// TIA Portal V16 export
// export: Created 2021-03-04T22:04:04.3689655Z, ExportSetting WithDefaults, DisplayName Totally Integrated Automation Portal, DisplayVersion V16, DisplayName TIA Portal Version Control Interface, DisplayVersion V16, DisplayName TIA Portal Openness, DisplayVersion V16, DisplayName SINAMICS Startdrive Advanced, DisplayVersion V16, DisplayName SINAMICS Startdrive G130, G150, S120, S150, SINAMICS MV, S210, DisplayVersion V16, DisplayName SINAMICS Startdrive G110M, G120, G120C, G120D, G120P, DisplayVersion V16, DisplayName STEP 7 Professional, DisplayVersion V16, DisplayName STEP 7 Safety, DisplayVersion V16, DisplayName WinCC Professional, DisplayVersion V16
VAR_GLOBAL   // PLC tag table "Library Constants"
END_VAR
VAR_GLOBAL CONSTANT   // user constants
   eSTATE_MANUAL : Int := 2;   // State Machine enumeration
   ePBLT_FLASHING_ENABLED : Int := 4;   // HMI PB LT enumeration
   eSTATE_RETRACTING : Int := 5;   // State Machine enumeration
   "IoScaling.S7Analog.Ni100.rScaledMax" : Real := 250.0;
   "IoScaling.S7Analog.Ni100.Climate.rScaledMax" : Real := 250.0;
   eSTEP_StoppingStart : Int := 4000;   // State Machine enumeration
   eSTEP_VerifyCenterComplete : Int := 7999;   // State Machine enumeration
   "IoScaling.S7Analog.150Ohms.rScaledMax" : Real := 150.0;
   "IoScaling.S7Analog.Default.bSwapBytes" : Bool := false;
   eANALOG_INPUTHIGHHIGH : Int := 102;
   eMOTION_DISABLED : Int := 4;   // Status Enumeration - Motion
   "IoScaling.S7Analog.Pt100.iRawMax" : Int := 8500;
   eSTEP_RetractingComplete : Int := 5999;   // State Machine enumeration
   eMODE_MANUAL : Int := 2;   // Mode enumeration
   eANALOG_INPUTINVALID : Int := 101;
   ePBLT_HIDDEN : Int := -1;   // HMI PB LT enumeration
   eVALVE_HOMEON : Int := 6;
   "IoScaling.S7Analog.Pt100.Climate.rScaledMin" : Real := -120.0;
   eHOME_ABS_RET_ABS : Int := 7;   // See MC_Home help for details
   eMOTION_ERROR : Int := 0;   // Status Enumeration - Motion
   ePB_MAINTAINED : Int := 1;   // HMI PB Type enumeration
   LKINCTRL_LENGTH_OF_PATHDATA_NAME : Int := 10;
   LKINCTRL_NO_OF_PATHDATA_ELEMENTS : Int := 15;
   "IoScaling.S7Analog.Pt100.Climate.iRawMax" : Int := 13000;
   eVALVE_ERROR : Int := 2;
   "IoScaling.S7Analog.Types.Pt100.Climate" : Int := 3;
   eMODE_INDEPENDENT : Int := 10;   // Mode
   "IoScaling.S7Analog.600Ohms.rScaledMax" : Real := 600.0;
   eMOTION_RUNNING : Int := 2;   // Status Enumeration - Motion
   "IoScaling.S7Analog.Ni100.Climate.rScaledMin" : Real := -60.0;
   eMOTION_STOPPED : Int := 1;   // Status Enumeration - Motion
   eMOTION_MAINTENANCE : Int := 3;   // Status Enumeration - Motion
   "IoScaling.S7Analog.Ni100.rScaledMin" : Real := -60.0;
   eSTATE_STOPPING : Int := 4;   // State Machine enumeration
   "IoScaling.S7Analog.Pt100.Climate.rScaledMax" : Real := 130.0;
   "IoScaling.S7Analog.Pt100.rScaledMax" : Real := 850.0;
   "IoScaling.S7Analog.Types.Ni100.Climate" : Int := 5;
   ePB_UNLATCH : Int := 3;   // HMI PB Type enumeration
   "IoScaling.S7Analog.Ni100.Climate.iRawMax" : Int := 25000;
   eSTEP_BladeChangeStart : Int := 6000;   // State Machine enumeration
   "IoScaling.S7Analog.300Ohms.rScaledMin" : Real := 0.0;
   "IoScaling.S7Analog.Types.Pt100" : Int := 2;
   LKINCTRL_PI : LReal := 3.1415926535897932846264;
   eVALVE_WORKPOSITION : Int := 3;
   eCAM_SYNCDIRECTION_SHORTESTWAY : Int := 3;   // See MC_CamIn help for details
   "IoScaling.S7Analog.Types.+-V/mA" : Int := 1;
   ePBLT_FLASHING_DISABLED : Int := 5;   // HMI PB LT enumeration
   "IoScaling.S7Analog.150Ohms.rScaledMin" : Real := 0.0;
   eHOME_ACCEPT_CURRENT : Int := 11;   // Used when the configured and current encoders don't match
   LKINCTRL_NO_OF_START_EXECUTE_CMDS : Int := 5;
   ePBLT_TRANSITIONING : Int := 2;   // HMI PB LT enumeration
   SM_ACTIVE_DYNAMICS : Int := 0;
   eVALVE_WORKON : Int := 5;
   "IoScaling.S7Analog.+-V/mA.iRawMax" : Int := 27648;
   eSTATE_INITIALIZATION : Int := 1;   // State Machine enumeration
   LKINCTRL_NO_OF_PATHDATA_PREBUFFER_ELEMENTS : Int := 5;
   eHOME_ABS_RET_OFFSET : Int := 6;   // See MC_Home help for details
   eSTEP_BladeChangeComplete : Int := 6999;   // State Machine enumeration
   eSTEP_RunningComplete : Int := 3999;   // State Machine enumeration
   eANALOG_READY : Int := 100;
   ePBLT_ENABLED : Int := 1;   // HMI PB LT enumeration
   "IoScaling.S7Analog.Pt100.Climate.iRawMin" : Int := -12000;
   eSTATE_RUNNING : Int := 3;   // State Machine enumeration
   LKINCTRL_NO_OF_LAST_FLAG : Int := 15;
   "IoScaling.S7Analog.Ni100.iRawMax" : Int := 2500;
   "IoScaling.S7Analog.Types.Default" : Int := 0;
   eHOME_ACCEPT_CONFIG : Int := 12;   // Used when the configured and current encoders don't match
   eSTEP_RunningStart : Int := 3000;   // State Machine enumeration
   "IoScaling.S7Analog.Default.iRawMin" : Int := 0;
   ePBLT_ACTIVE : Int := 3;   // HMI PB LT enumeration
   "IoScaling.S7Analog.Types.Ni100" : Int := 4;
   eMODE_AUTO : Int := 1;   // Mode enumeration
   "IoScaling.S7Analog.Default.iRawMax" : Int := 27648;
   ePBLT_DISABLED : Int := 0;   // HMI PB LT enumeration
   LKINCTRL_NO_OF_SEQ_EXECUTE_CMDS : Int := 5;
   eSTEP_StoppingComplete : Int := 4999;   // State Machine enumeration
   "IoScaling.S7Analog.Ni100.Climate.iRawMin" : Int := -6000;
   "IoScaling.S7Analog.Pt100.iRawMin" : Int := -2000;
   ePB_LATCH : Int := 2;   // HMI PB Type enumeration
   eVALVE_ESTOP : Int := 1;
   eSTEP_RetractingStart : Int := 5000;   // State Machine enumeration
   "IoScaling.S7Analog.300Ohms.rScaledMax" : Real := 300.0;
   eANALOG_INPUTLOW : Int := 105;
   "IoScaling.S7Analog.Pt100.rScaledMin" : Real := -200.0;
   eSTATE_BLADECHANGE : Int := 6;   // State Machine enumeration
   "IoScaling.S7Analog.600Ohms.rScaledMin" : Real := 0.0;
   eSTATE_VERIFYCENTER : Int := 7;   // State Machine enumeration
   eVALVE_STOPPED : Int := 0;
   eCAM_SYNCPROFILEREFERENCE_LEADINGVALUEDISTANCE : Int := 1;   // See MC_CamIn help for details
   "IoScaling.S7Analog.Ni100.iRawMin" : Int := -600;
   ePB_HELD : Int := 4;   // HMI PB Type enumeration
   LKINCTRL_NO_OF_CMD_SETFLAGS : Int := 8;
   eSTEP_VerifyCenterStart : Int := 7000;   // State Machine enumeration
   eVALVE_HOMEPOSITION : Int := 4;
   eANALOG_INPUTHIGH : Int := 104;
   eANALOG_INPUTLOWLOW : Int := 103;
   "IoScaling.S7Analog.+-V/mA.iRawMin" : Int := -27648;
   ePB_MOMENTARY : Int := 0;   // HMI PB Type enumeration
   "Modes.PID.Pretuning" : Int := 1;
   "TotalizerTimeUnits.DAYS" : Int := 4;
   "HMI.Status.ForwardWork" : Int := 3;
   "FIFO.iQueueDisabled" : Int := -1;
   "Handshakes.iSize" : Int := 5;
   "Modes.Auto" : Int := 1;
   "HMI.Status.Generic1" : Int := 101;
   "Simocode.Types.DirectStarter" : Int := 1;
   "Estop.MinSetPoint" : Int := 0;
   "Simocode.Types.OverloadRelay" : Int := 0;
   "HMI.Status.SimulatedReverseHome" : Int := 8;
   "TotalizerTimeUnits.MILLISECONDS" : Int := 0;
   "HMI.Status.Generic4" : Int := 104;
   "SoftStarter.HMI.Status.EStop" : Int := 1;
   "HMI.Status.OnForwardWork" : Int := 5;
   "DataTypes.iMaxInt" : Int := 32767;
   "FIFO.iQueueSize" : Int := 5;
   "Modes.PID.ManualMode" : Int := 4;
   "TotalizerTimeUnits.SECONDS" : Int := 1;
   "SoftStarter.Types.3RW30" : Int := 30;
   "HMI.Status.Generic3" : Int := 103;
   "HMI.Status.OnReverseHome" : Int := 6;
   "HMI.Status.Estop" : Int := 1;
   "SoftStarter.HMI.Status.Error" : Int := 2;
   "HMI.Status.Generic6" : Int := 106;
   "DataTypes.rMaxReal" : Real := 3.402823e38;
   "SoftStarter.HMI.Status.Off" : Int := 0;
   "Modes.PID.Inactive" : Int := 0;
   "HMI.Status.GenericNone" : Int := 100;
   "HMI.Status.Generic2" : Int := 102;
   "Modes.PID.AutoMode" : Int := 3;
   "SoftStarter.HMI.Status.On" : Int := 4;
   "Estop.HMISetPoint" : Int := 2;
   "HMI.Status.ReverseHome" : Int := 4;
   "DataTypes.rMinReal" : Real := -3.402823e38;
   "TotalizerTimeUnits.MINUTES" : Int := 2;
   "Modes.PID.FineTuning" : Int := 2;
   "TotalizerTimeUnits.HOURS" : Int := 3;
   "Ramp.Timed" : Int := 1;
   "Estop.MaxSetPoint" : Int := 1;
   "SoftStarter.Types.3RW40" : Int := 40;
   "Ramp.Continuous" : Int := 0;
   "HMI.Status.Generic5" : Int := 105;
   "Modes.Manual" : Int := 2;
   "Modes.Stop" : Int := 0;
   "HMI.Status.SimulatedOnReverseHome" : Int := 10;
   "Simocode.Types.ReversingStarter" : Int := 2;
   "Modes.Independent" : Int := 10;
   "DataTypes.iMinInt" : Int := -32768;
   "SoftStarter.HMI.Status.RampUp" : Int := 3;
   "SoftStarter.HMI.Status.RampDown" : Int := 5;
   "HMI.Status.Error" : Int := 2;
   "HMI.Status.SimulatedOnForwardWork" : Int := 9;
   "HMI.Status.SimulatedForwardWork" : Int := 7;
   "HMI.Status.Stopped" : Int := 0;
END_VAR
